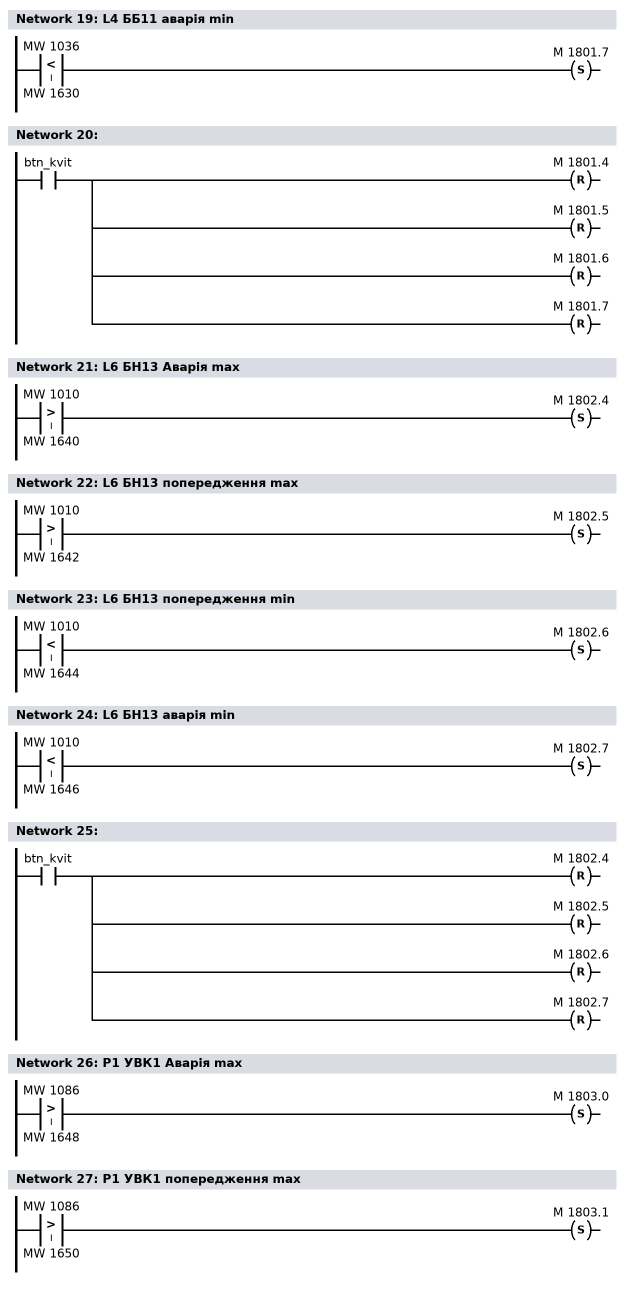
NETWORK
TITLE = L4 ББ11 аварія min
      L     MW 1036;
      L     MW 1630;
      <I;
      S     M 1801.7;
NETWORK
TITLE =
      A     "btn_kvit";
      R     M 1801.4;
      R     M 1801.5;
      R     M 1801.6;
      R     M 1801.7;
NETWORK
TITLE = L6 БН13 Аварія max
//*************************************************
      L     MW 1010;
      L     MW 1640;
      >I;
      S     M 1802.4;
NETWORK
TITLE = L6 БН13 попередження max
      L     MW 1010;
      L     MW 1642;
      >I;
      S     M 1802.5;
NETWORK
TITLE = L6 БН13 попередження min
      L     MW 1010;
      L     MW 1644;
      <I;
      S     M 1802.6;
NETWORK
TITLE = L6 БН13 аварія min
      L     MW 1010;
      L     MW 1646;
      <I;
      S     M 1802.7;
NETWORK
TITLE =
      A     "btn_kvit";
      R     M 1802.4;
      R     M 1802.5;
      R     M 1802.6;
      R     M 1802.7;
NETWORK
TITLE = P1 УВК1 Аварія max
//*************************************************
      L     MW 1086;
      L     MW 1648;
      >I;
      S     M 1803.0;
NETWORK
TITLE = P1 УВК1 попередження max
      L     MW 1086;
      L     MW 1650;
      >I;
      S     M 1803.1;
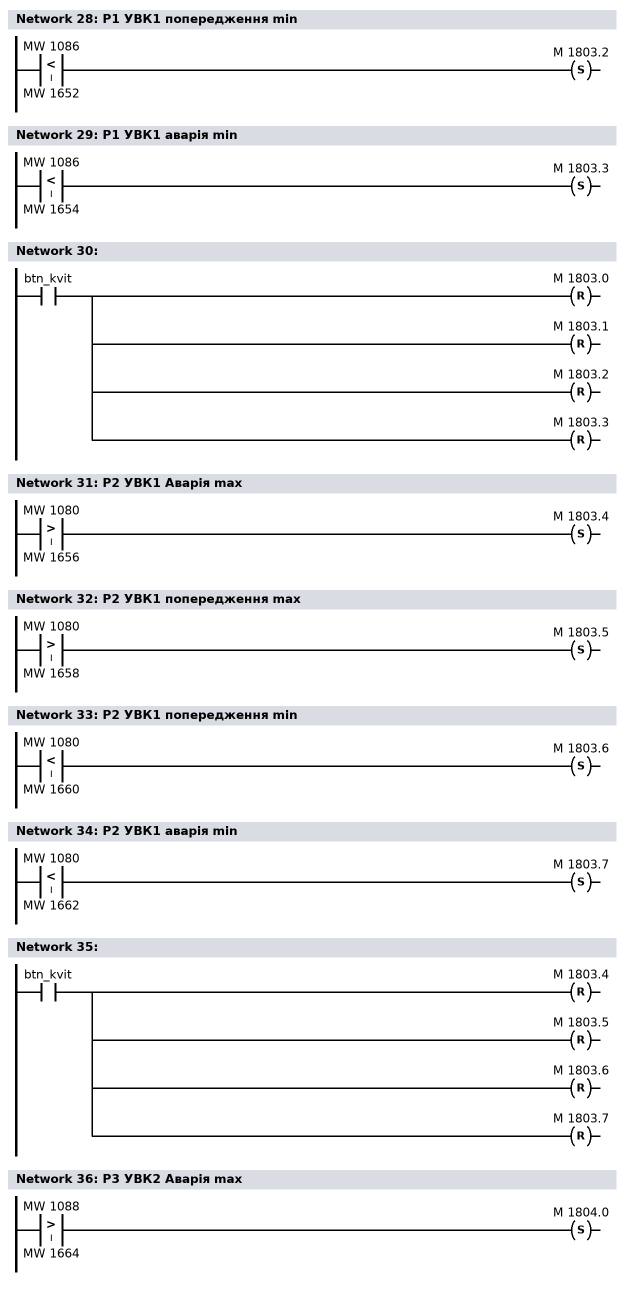
NETWORK
TITLE = P1 УВК1 попередження min
      L     MW 1086;
      L     MW 1652;
      <I;
      S     M 1803.2;
NETWORK
TITLE = P1 УВК1 аварія min
      L     MW 1086;
      L     MW 1654;
      <I;
      S     M 1803.3;
NETWORK
TITLE =
      A     "btn_kvit";
      R     M 1803.0;
      R     M 1803.1;
      R     M 1803.2;
      R     M 1803.3;
NETWORK
TITLE = P2 УВК1 Аварія max
//*************************************************
      L     MW 1080;
      L     MW 1656;
      >I;
      S     M 1803.4;
NETWORK
TITLE = P2 УВК1 попередження max
      L     MW 1080;
      L     MW 1658;
      >I;
      S     M 1803.5;
NETWORK
TITLE = P2 УВК1 попередження min
      L     MW 1080;
      L     MW 1660;
      <I;
      S     M 1803.6;
NETWORK
TITLE = P2 УВК1 аварія min
      L     MW 1080;
      L     MW 1662;
      <I;
      S     M 1803.7;
NETWORK
TITLE =
      A     "btn_kvit";
      R     M 1803.4;
      R     M 1803.5;
      R     M 1803.6;
      R     M 1803.7;
NETWORK
TITLE = P3 УВК2 Аварія max
//*************************************************
      L     MW 1088;
      L     MW 1664;
      >I;
      S     M 1804.0;
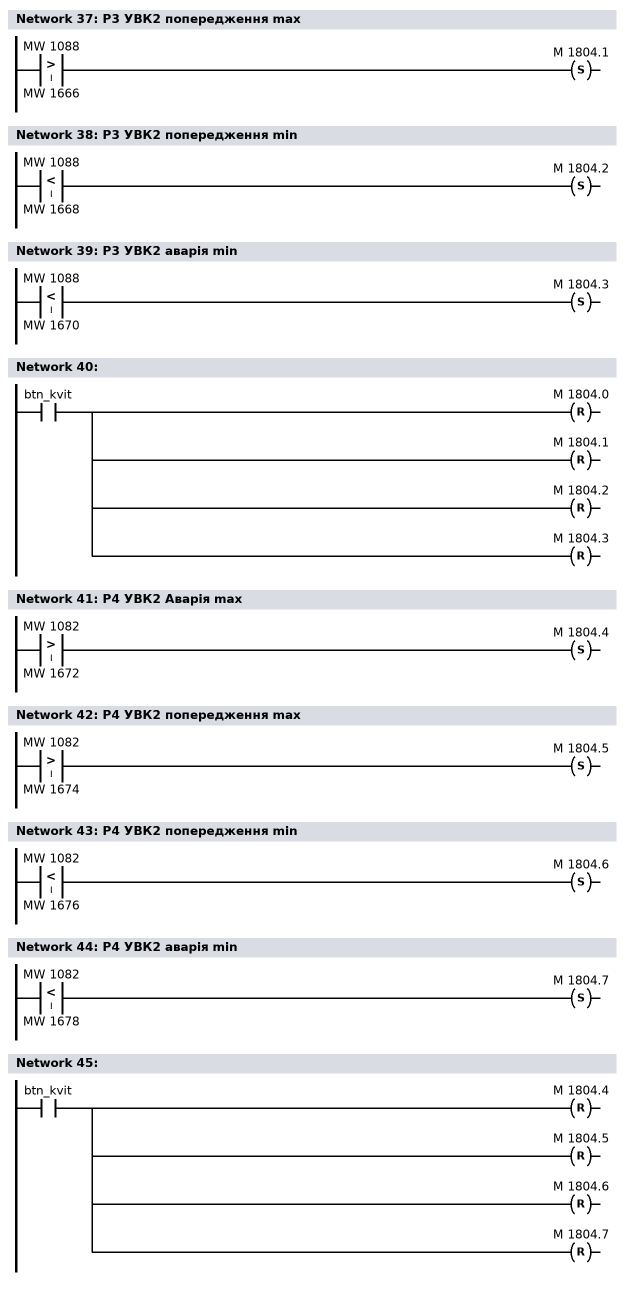
NETWORK
TITLE = P3 УВК2 попередження max
      L     MW 1088;
      L     MW 1666;
      >I;
      S     M 1804.1;
NETWORK
TITLE = P3 УВК2 попередження min
      L     MW 1088;
      L     MW 1668;
      <I;
      S     M 1804.2;
NETWORK
TITLE = P3 УВК2 аварія min
      L     MW 1088;
      L     MW 1670;
      <I;
      S     M 1804.3;
NETWORK
TITLE =
      A     "btn_kvit";
      R     M 1804.0;
      R     M 1804.1;
      R     M 1804.2;
      R     M 1804.3;
NETWORK
TITLE = P4 УВК2 Аварія max
//*************************************************
      L     MW 1082;
      L     MW 1672;
      >I;
      S     M 1804.4;
NETWORK
TITLE = P4 УВК2 попередження max
      L     MW 1082;
      L     MW 1674;
      >I;
      S     M 1804.5;
NETWORK
TITLE = P4 УВК2 попередження min
      L     MW 1082;
      L     MW 1676;
      <I;
      S     M 1804.6;
NETWORK
TITLE = P4 УВК2 аварія min
      L     MW 1082;
      L     MW 1678;
      <I;
      S     M 1804.7;
NETWORK
TITLE =
      A     "btn_kvit";
      R     M 1804.4;
      R     M 1804.5;
      R     M 1804.6;
      R     M 1804.7;
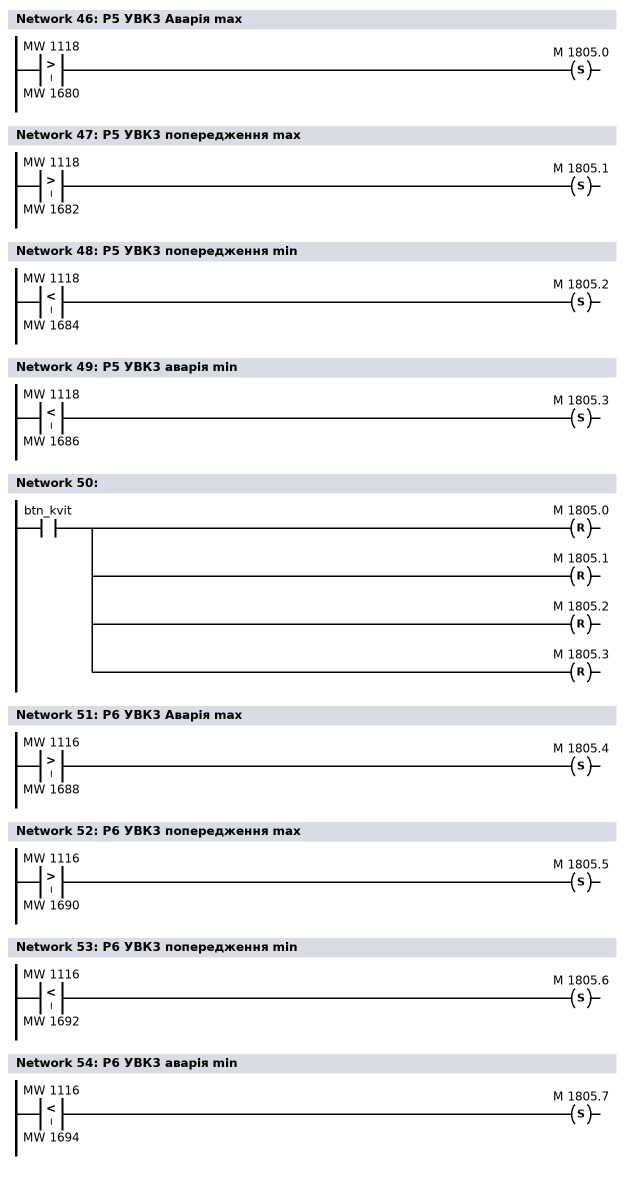
NETWORK
TITLE = P5 УВК3 Аварія max
//*************************************************
      L     MW 1118;
      L     MW 1680;
      >I;
      S     M 1805.0;
NETWORK
TITLE = P5 УВК3 попередження max
      L     MW 1118;
      L     MW 1682;
      >I;
      S     M 1805.1;
NETWORK
TITLE = P5 УВК3 попередження min
      L     MW 1118;
      L     MW 1684;
      <I;
      S     M 1805.2;
NETWORK
TITLE = P5 УВК3 аварія min
      L     MW 1118;
      L     MW 1686;
      <I;
      S     M 1805.3;
NETWORK
TITLE =
      A     "btn_kvit";
      R     M 1805.0;
      R     M 1805.1;
      R     M 1805.2;
      R     M 1805.3;
NETWORK
TITLE = P6 УВК3 Аварія max
//*************************************************
      L     MW 1116;
      L     MW 1688;
      >I;
      S     M 1805.4;
NETWORK
TITLE = P6 УВК3 попередження max
      L     MW 1116;
      L     MW 1690;
      >I;
      S     M 1805.5;
NETWORK
TITLE = P6 УВК3 попередження min
      L     MW 1116;
      L     MW 1692;
      <I;
      S     M 1805.6;
NETWORK
TITLE = P6 УВК3 аварія min
      L     MW 1116;
      L     MW 1694;
      <I;
      S     M 1805.7;
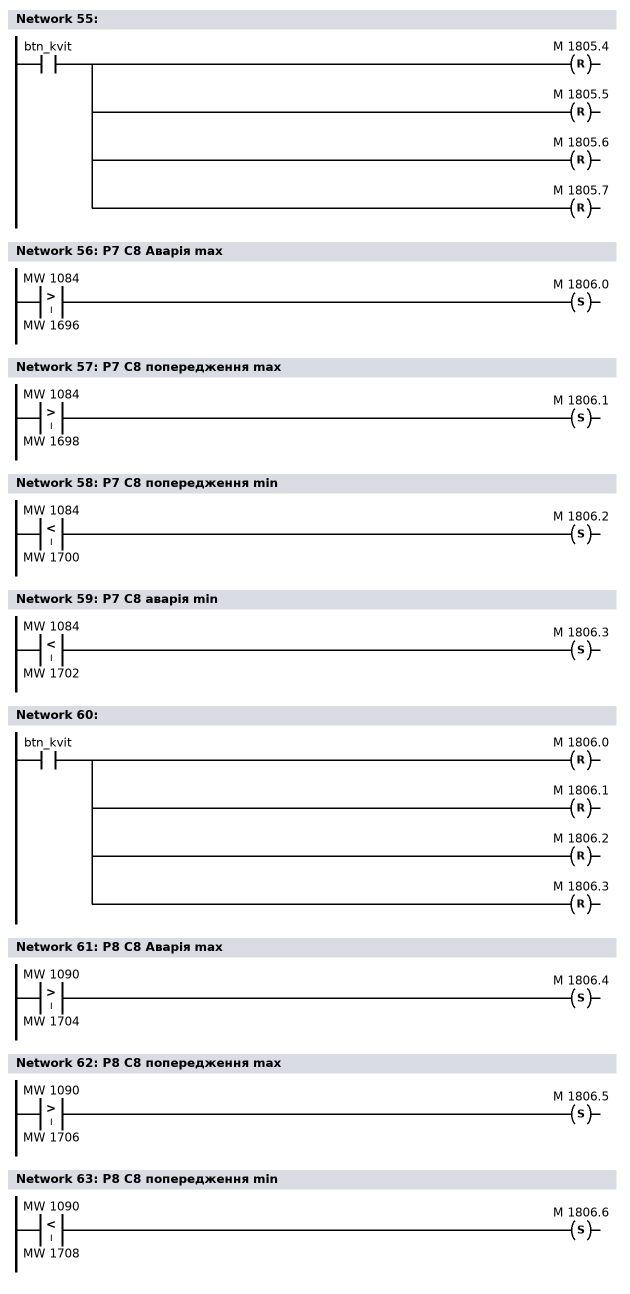
NETWORK
TITLE =
      A     "btn_kvit";
      R     M 1805.4;
      R     M 1805.5;
      R     M 1805.6;
      R     M 1805.7;
NETWORK
TITLE = P7 С8 Аварія max
//*************************************************
      L     MW 1084;
      L     MW 1696;
      >I;
      S     M 1806.0;
NETWORK
TITLE = P7 С8 попередження max
      L     MW 1084;
      L     MW 1698;
      >I;
      S     M 1806.1;
NETWORK
TITLE = P7 С8 попередження min
      L     MW 1084;
      L     MW 1700;
      <I;
      S     M 1806.2;
NETWORK
TITLE = P7 С8 аварія min
      L     MW 1084;
      L     MW 1702;
      <I;
      S     M 1806.3;
NETWORK
TITLE =
      A     "btn_kvit";
      R     M 1806.0;
      R     M 1806.1;
      R     M 1806.2;
      R     M 1806.3;
NETWORK
TITLE = P8 С8 Аварія max
//*************************************************
      L     MW 1090;
      L     MW 1704;
      >I;
      S     M 1806.4;
NETWORK
TITLE = P8 С8 попередження max
      L     MW 1090;
      L     MW 1706;
      >I;
      S     M 1806.5;
NETWORK
TITLE = P8 С8 попередження min
      L     MW 1090;
      L     MW 1708;
      <I;
      S     M 1806.6;
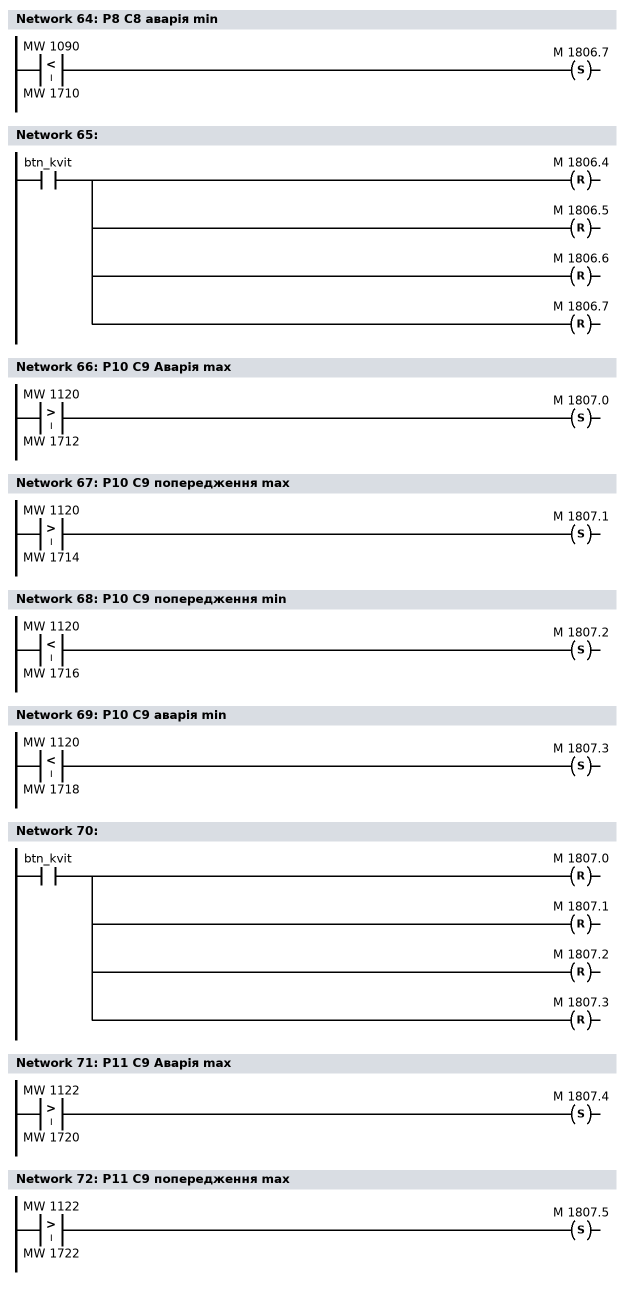
NETWORK
TITLE = P8 С8 аварія min
      L     MW 1090;
      L     MW 1710;
      <I;
      S     M 1806.7;
NETWORK
TITLE =
      A     "btn_kvit";
      R     M 1806.4;
      R     M 1806.5;
      R     M 1806.6;
      R     M 1806.7;
NETWORK
TITLE = P10 С9 Аварія max
//*************************************************
      L     MW 1120;
      L     MW 1712;
      >I;
      S     M 1807.0;
NETWORK
TITLE = P10 С9 попередження max
      L     MW 1120;
      L     MW 1714;
      >I;
      S     M 1807.1;
NETWORK
TITLE = P10 С9 попередження min
      L     MW 1120;
      L     MW 1716;
      <I;
      S     M 1807.2;
NETWORK
TITLE = P10 С9 аварія min
      L     MW 1120;
      L     MW 1718;
      <I;
      S     M 1807.3;
NETWORK
TITLE =
      A     "btn_kvit";
      R     M 1807.0;
      R     M 1807.1;
      R     M 1807.2;
      R     M 1807.3;
NETWORK
TITLE = P11 С9 Аварія max
//*************************************************
      L     MW 1122;
      L     MW 1720;
      >I;
      S     M 1807.4;
NETWORK
TITLE = P11 С9 попередження max
      L     MW 1122;
      L     MW 1722;
      >I;
      S     M 1807.5;
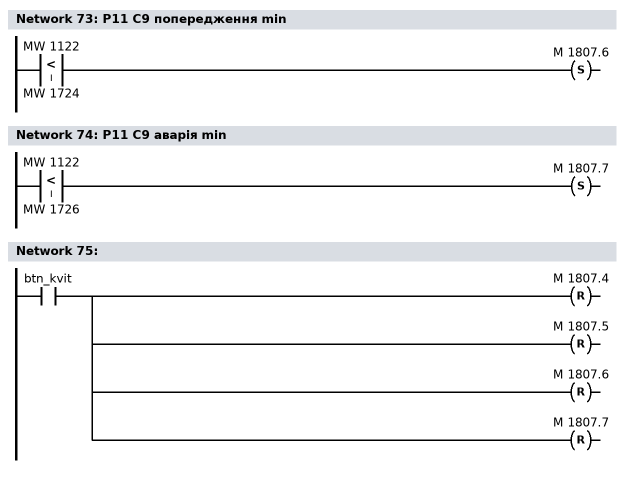
NETWORK
TITLE = P11 С9 попередження min
      L     MW 1122;
      L     MW 1724;
      <I;
      S     M 1807.6;
NETWORK
TITLE = P11 С9 аварія min
      L     MW 1122;
      L     MW 1726;
      <I;
      S     M 1807.7;
NETWORK
TITLE =
      A     "btn_kvit";
      R     M 1807.4;
      R     M 1807.5;
      R     M 1807.6;
      R     M 1807.7;
END_FUNCTION_BLOCK

// FB 58: know-how protected block, not included

FUNCTION "DO_MANUAL" : VOID	// FC 1
VERSION : 0.1
VAR_INPUT
  MANUAL : BOOL ;
  PUSK : BOOL ;
  STOP : BOOL ;
END_VAR
VAR_OUTPUT
  M_DO : BOOL ;
END_VAR
BEGIN
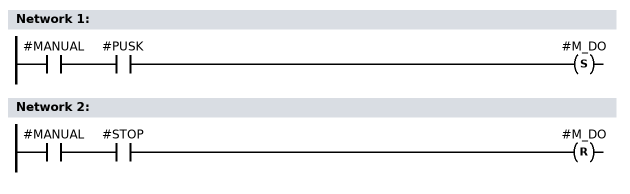
NETWORK
TITLE =
      A     #MANUAL;
      A     #PUSK;
      S     #M_DO;
NETWORK
TITLE =
      A     #MANUAL;
      A     #STOP;
      R     #M_DO;
END_FUNCTION

// FC 105: know-how protected block, not included

// FC 106: know-how protected block, not included

DATA_BLOCK DB 2
VERSION : 0.1
"MD_to_MW"
BEGIN
END_DATA_BLOCK

DATA_BLOCK DB 3
VERSION : 0.0
"DO_Control"
BEGIN
END_DATA_BLOCK

DATA_BLOCK DB 4
VERSION : 0.1
"DI_DO_STATE"
BEGIN
END_DATA_BLOCK

DATA_BLOCK DB 6
VERSION : 0.0
"dat_alm"
BEGIN
END_DATA_BLOCK

DATA_BLOCK DB 14
AUTHOR : SIMATIC
FAMILY : COM_FUNC
VERSION : 0.0
"GET"
BEGIN
END_DATA_BLOCK

DATA_BLOCK "COM"	// DB 100
VERSION : 0.1
  STRUCT
   dZN1_cur : REAL ;
   dUVK_nas1_cur : REAL ;
   dUVK_nas2_cur : REAL ;
   dUZ1_in : REAL ;
   dUZ1_out : REAL ;
   dPidsit_riv : REAL ;
   dVak_suknom1 : REAL ;
   dVak_suknom2 : REAL ;
   dVak_suknom3 : REAL ;
   dVak_suknom4 : REAL ;
   dVak_suknom5 : REAL ;
   dVak_suknom6 : REAL ;
   dVak_val1 : REAL ;
   dVak_val2 : REAL ;
   dVak_mok1 : REAL ;
   dVak_mok2 : REAL ;
   dVak_mok3 : REAL ;
   dVak_mok4 : REAL ;
   dVak_suh1 : REAL ;
   dVak_suh2 : REAL ;
   dVak_suh3 : REAL ;
   dVak_suh4 : REAL ;
   dVak_suh5 : REAL ;
   dVak_suh6 : REAL ;
   dVak_VN1 : REAL ;
   dVak_VN2 : REAL ;
   dVak_VN3 : REAL ;
   dVak_VN4 : REAL ;
   dVak_VN5 : REAL ;
   dBM8_riv : REAL ;
   dBO9_riv : REAL ;
   dBZ10_riv : REAL ;
   dBB11_riv : REAL ;
   dGauch_riv : REAL ;
   dNC32_riv : REAL ;
   dNC35_riv : REAL ;
   dPriamok_riv : REAL ;
   dGRG_riv : REAL ;
   task_ZNM12_re : REAL ;
   task_ZNM15_re : REAL ;
   dUVK1_in : REAL ;
   dUVK2_in : REAL ;
   dC8_in : REAL ;
   dUVK1_out : REAL ;
   dUVK2_out : REAL ;
   dC8_out : REAL ;
   dSUM_Pr_nya : REAL ;
   dConc1_nya : REAL ;
   dRiv_Skop : REAL ;
   dRiv_Bak_pid_nya : REAL ;
   dPr_uzloulov_in : REAL ;
   dMlyn_in : REAL ;
   dRiv_Bak_nap : REAL ;
   dMlyn_out : REAL ;
   dPr_uzloulov_out : REAL ;
   dRIV_NYA : REAL ;
  END_STRUCT ;	
BEGIN
END_DATA_BLOCK

DATA_BLOCK DB 101
VERSION : 0.0
"Dat_Filt"
BEGIN
END_DATA_BLOCK

DATA_BLOCK DB 102
VERSION : 0.0
"Dat_Filt"
BEGIN
END_DATA_BLOCK

DATA_BLOCK DB 103
VERSION : 0.0
"Dat_Filt"
BEGIN
END_DATA_BLOCK

DATA_BLOCK DB 104
VERSION : 0.0
"Dat_Filt"
BEGIN
END_DATA_BLOCK

DATA_BLOCK DB 105
VERSION : 0.0
"Dat_Filt"
BEGIN
END_DATA_BLOCK

DATA_BLOCK DB 106
VERSION : 0.0
"Dat_Filt"
BEGIN
END_DATA_BLOCK

DATA_BLOCK DB 107
VERSION : 0.0
"Dat_Filt"
BEGIN
END_DATA_BLOCK

DATA_BLOCK DB 108
VERSION : 0.0
"Dat_Filt"
BEGIN
END_DATA_BLOCK

DATA_BLOCK DB 109
VERSION : 0.0
"Dat_Filt"
BEGIN
END_DATA_BLOCK

DATA_BLOCK DB 110
VERSION : 0.0
"Dat_Filt"
BEGIN
END_DATA_BLOCK

DATA_BLOCK DB 111
VERSION : 0.0
"Dat_Filt"
BEGIN
END_DATA_BLOCK

DATA_BLOCK DB 112
VERSION : 0.0
"Dat_Filt"
BEGIN
END_DATA_BLOCK

DATA_BLOCK DB 113
VERSION : 0.0
"Dat_Filt"
BEGIN
END_DATA_BLOCK

DATA_BLOCK DB 114
VERSION : 0.0
"Dat_Filt"
BEGIN
END_DATA_BLOCK

DATA_BLOCK DB 115
VERSION : 0.0
"Dat_Filt"
BEGIN
END_DATA_BLOCK

DATA_BLOCK DB 116
VERSION : 0.0
"Dat_Filt"
BEGIN
END_DATA_BLOCK

DATA_BLOCK DB 117
VERSION : 0.0
"Dat_Filt"
BEGIN
END_DATA_BLOCK

DATA_BLOCK DB 118
VERSION : 0.0
"Dat_Filt"
BEGIN
END_DATA_BLOCK

DATA_BLOCK DB 119
VERSION : 0.0
"Dat_Filt"
BEGIN
END_DATA_BLOCK

DATA_BLOCK DB 120
VERSION : 0.0
"Dat_Filt"
BEGIN
END_DATA_BLOCK

DATA_BLOCK DB 121
VERSION : 0.0
"Dat_Filt"
BEGIN
END_DATA_BLOCK

DATA_BLOCK DB 122
VERSION : 0.0
"Dat_Filt"
BEGIN
END_DATA_BLOCK

DATA_BLOCK DB 123
VERSION : 0.0
"Dat_Filt"
BEGIN
END_DATA_BLOCK

DATA_BLOCK DB 124
VERSION : 0.0
"Dat_Filt"
BEGIN
END_DATA_BLOCK

DATA_BLOCK DB 125
VERSION : 0.0
"Dat_Filt"
BEGIN
END_DATA_BLOCK

DATA_BLOCK DB 126
VERSION : 0.0
"Dat_Filt"
BEGIN
END_DATA_BLOCK

DATA_BLOCK DB 127
VERSION : 0.0
"Dat_Filt"
BEGIN
END_DATA_BLOCK

DATA_BLOCK DB 128
VERSION : 0.0
"Dat_Filt"
BEGIN
END_DATA_BLOCK

DATA_BLOCK DB 141
VERSION : 0.0
"Dat_Filt"
BEGIN
END_DATA_BLOCK

DATA_BLOCK DB 142
VERSION : 0.0
"Dat_Filt"
BEGIN
END_DATA_BLOCK

DATA_BLOCK DB 143
VERSION : 0.0
"Dat_Filt"
BEGIN
END_DATA_BLOCK

DATA_BLOCK DB 144
VERSION : 0.0
"Dat_Filt"
BEGIN
END_DATA_BLOCK

DATA_BLOCK DB 145
VERSION : 0.0
"Dat_Filt"
BEGIN
END_DATA_BLOCK

DATA_BLOCK DB 146
VERSION : 0.0
"Dat_Filt"
BEGIN
END_DATA_BLOCK

DATA_BLOCK DB 147
VERSION : 0.0
"Dat_Filt"
BEGIN
END_DATA_BLOCK

DATA_BLOCK DB 148
VERSION : 0.0
"Dat_Filt"
BEGIN
END_DATA_BLOCK

DATA_BLOCK DB 149
VERSION : 0.0
"Dat_Filt"
BEGIN
END_DATA_BLOCK

DATA_BLOCK DB 150
VERSION : 0.0
"Dat_Filt"
BEGIN
END_DATA_BLOCK

DATA_BLOCK DB 151
VERSION : 0.0
"Dat_Filt"
BEGIN
END_DATA_BLOCK

DATA_BLOCK DB 152
VERSION : 0.0
"Dat_Filt"
BEGIN
END_DATA_BLOCK

DATA_BLOCK DB 153
VERSION : 0.0
"Dat_Filt"
BEGIN
END_DATA_BLOCK

DATA_BLOCK DB 154
VERSION : 0.0
"Dat_Filt"
BEGIN
END_DATA_BLOCK

DATA_BLOCK DB 155
VERSION : 0.0
"Dat_Filt"
BEGIN
END_DATA_BLOCK

DATA_BLOCK DB 300
VERSION : 0.0
"PID_AO_control"
BEGIN
END_DATA_BLOCK

DATA_BLOCK DB 301
VERSION : 0.0
"PID_AO_control"
BEGIN
END_DATA_BLOCK

DATA_BLOCK DB 302
VERSION : 0.0
"PID_AO_control"
BEGIN
END_DATA_BLOCK

DATA_BLOCK "znm15_pid"	// DB 500
AUTHOR : SIMATIC
FAMILY : CONTROL
VERSION : 0.0
"TCONT_CP"
BEGIN
END_DATA_BLOCK

DATA_BLOCK "CV_dConc1_pid"	// DB 501
AUTHOR : SIMATIC
FAMILY : CONTROL
VERSION : 0.0
"TCONT_CP"
BEGIN
END_DATA_BLOCK

DATA_BLOCK "zadv_riv_nya"	// DB 502
AUTHOR : SIMATIC
FAMILY : CONTROL
VERSION : 0.0
"TCONT_CP"
BEGIN
END_DATA_BLOCK

ORGANIZATION_BLOCK "CYCL_EXC"	// OB 1
TITLE = "Main Program Sweep (Cycle)"
VERSION : 0.1
VAR_TEMP
  OB1_EV_CLASS : BYTE ;	//Bits 0-3 = 1 (Coming event), Bits 4-7 = 1 (Event class 1)
  OB1_SCAN_1 : BYTE ;	//1 (Cold restart scan 1 of OB 1), 3 (Scan 2-n of OB 1)
  OB1_PRIORITY : BYTE ;	//Priority of OB Execution
  OB1_OB_NUMBR : BYTE ;	//1 (Organization block 1, OB1)
  OB1_RESERVED_1 : BYTE ;	//Reserved for system
  OB1_RESERVED_2 : BYTE ;	//Reserved for system
  OB1_PREV_CYCLE : INT ;	//Cycle time of previous OB1 scan (milliseconds)
  OB1_MIN_CYCLE : INT ;	//Minimum cycle time of OB1 (milliseconds)
  OB1_MAX_CYCLE : INT ;	//Maximum cycle time of OB1 (milliseconds)
  OB1_DATE_TIME : DATE_AND_TIME ;	//Date and time OB1 started
  err_ZN1_cur : BOOL ;
  err_UVK1_cur : BOOL ;
  err_UVK2_cur : BOOL ;
  err_UZ1_in : BOOL ;
  err_UZ1_out : BOOL ;
  err_pidsit_riv : BOOL ;
  err_vak_suknom1 : BOOL ;
  err_vak_suknom2 : BOOL ;
  err_vak_suknom3 : BOOL ;
  err_vak_suknom4 : BOOL ;
  err_vak_suknom5 : BOOL ;
  err_vak_suknom6 : BOOL ;
  err_vak_val1 : BOOL ;
  err_vak_val2 : BOOL ;
  err_vak_mok1 : BOOL ;
  err_vak_mok2 : BOOL ;
  err_vak_mok3 : BOOL ;
  err_vak_mok4 : BOOL ;
  err_suh1 : BOOL ;
  err_suh2 : BOOL ;
  err_suh3 : BOOL ;
  err_suh4 : BOOL ;
  err_suh5 : BOOL ;
  err_suh6 : BOOL ;
  err_vak_VN1 : BOOL ;
  err_vak_VN2 : BOOL ;
  err_vak_VN3 : BOOL ;
  err_vak_VN4 : BOOL ;
  err_vak_VN5 : BOOL ;
  err_BM8_riv : BOOL ;
  err_BO9_riv : BOOL ;
  err_BZ10_riv : BOOL ;
  err_BB11_riv : BOOL ;
  err_Gauch_riv : BOOL ;
  err_NC32_riv : BOOL ;
  err_NC35_riv : BOOL ;
  err_Priamok_riv : BOOL ;
  err_GRG_riv : BOOL ;
  ZNM12_ret : WORD ;
  ZNM15_ret : WORD ;
  bipolar : BOOL ;
  err_dUVK1in : BOOL ;
  err_dUVK2in : BOOL ;
  err_dC8in : BOOL ;
  err_dUVK1out : BOOL ;
  err_dUVK2out : BOOL ;
  err_dC8out : BOOL ;
  err_dSumPR : BOOL ;
  err_dConc1 : BOOL ;
  err_dBakSkop : BOOL ;
  err_dBakpidNya : BOOL ;
  err_dMlyn_in : BOOL ;
  err_uzloulov_in : BOOL ;
  err_dMlyn_out : BOOL ;
  err_uzloulov_out : BOOL ;
  bypass : BOOL ;
  err_dRIV_NYA : BOOL ;
END_VAR
BEGIN
NETWORK
TITLE = Из ПЛК ДВГ берем 10 байт в ПЛК КИП (кнопки "ручний режим")
      A     M 100.3;
      =     L 33.0;
      BLD   103;
      BLD   9;
      =     L 38.0;
      CDB;
      OPN   DI 14;
      TAR2  LD 34;
      A     L 33.0;
      =     DIX 0.0;
      L     2;
      T     DIW 2;
      L     W#16#1002;
      T     DIW 8;
      L     10;
      T     DIW 10;
      L     0;
      T     DIW 12;
      L     P#M 2000.0;
      T     DID 14;
      L     W#16#1002;
      T     DIW 48;
      L     10;
      T     DIW 50;
      L     0;
      T     DIW 52;
      L     P#M 6000.0;
      T     DID 54;
      LAR2  P#DBX 0.0;
      UC    "GET";
      LAR2  LD 34;
      CDB;
      BLD   10;
      NOP   0;
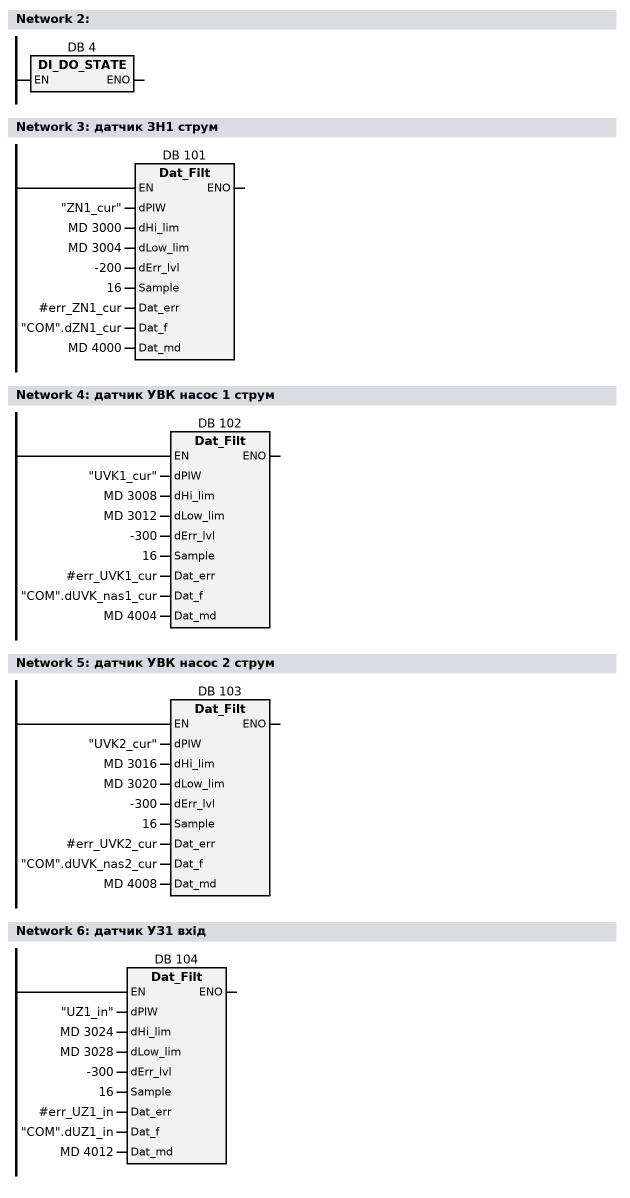
NETWORK
TITLE =
      CALL  "DI_DO_STATE" , DB 4;
      NOP   0;
NETWORK
TITLE = датчик ЗН1 струм  
      CALL  "Dat_Filt" , DB 101 (
           dPIW                     := "ZN1_cur",
           dHi_lim                  := MD 3000,
           dLow_lim                 := MD 3004,
           dErr_lvl                 := -200,
           Sample                   := 16,
           Dat_err                  := #err_ZN1_cur,
           Dat_f                    := "COM".dZN1_cur,
           Dat_md                   := MD 4000);
      NOP   0;
NETWORK
TITLE = датчик УВК насос 1 струм 
      CALL  "Dat_Filt" , DB 102 (
           dPIW                     := "UVK1_cur",
           dHi_lim                  := MD 3008,
           dLow_lim                 := MD 3012,
           dErr_lvl                 := -300,
           Sample                   := 16,
           Dat_err                  := #err_UVK1_cur,
           Dat_f                    := "COM".dUVK_nas1_cur,
           Dat_md                   := MD 4004);
      NOP   0;
NETWORK
TITLE = датчик УВК насос 2 струм 
      CALL  "Dat_Filt" , DB 103 (
           dPIW                     := "UVK2_cur",
           dHi_lim                  := MD 3016,
           dLow_lim                 := MD 3020,
           dErr_lvl                 := -300,
           Sample                   := 16,
           Dat_err                  := #err_UVK2_cur,
           Dat_f                    := "COM".dUVK_nas2_cur,
           Dat_md                   := MD 4008);
      NOP   0;
NETWORK
TITLE = датчик УЗ1 вхід
      CALL  "Dat_Filt" , DB 104 (
           dPIW                     := "UZ1_in",
           dHi_lim                  := MD 3024,
           dLow_lim                 := MD 3028,
           dErr_lvl                 := -300,
           Sample                   := 16,
           Dat_err                  := #err_UZ1_in,
           Dat_f                    := "COM".dUZ1_in,
           Dat_md                   := MD 4012);
      NOP   0;
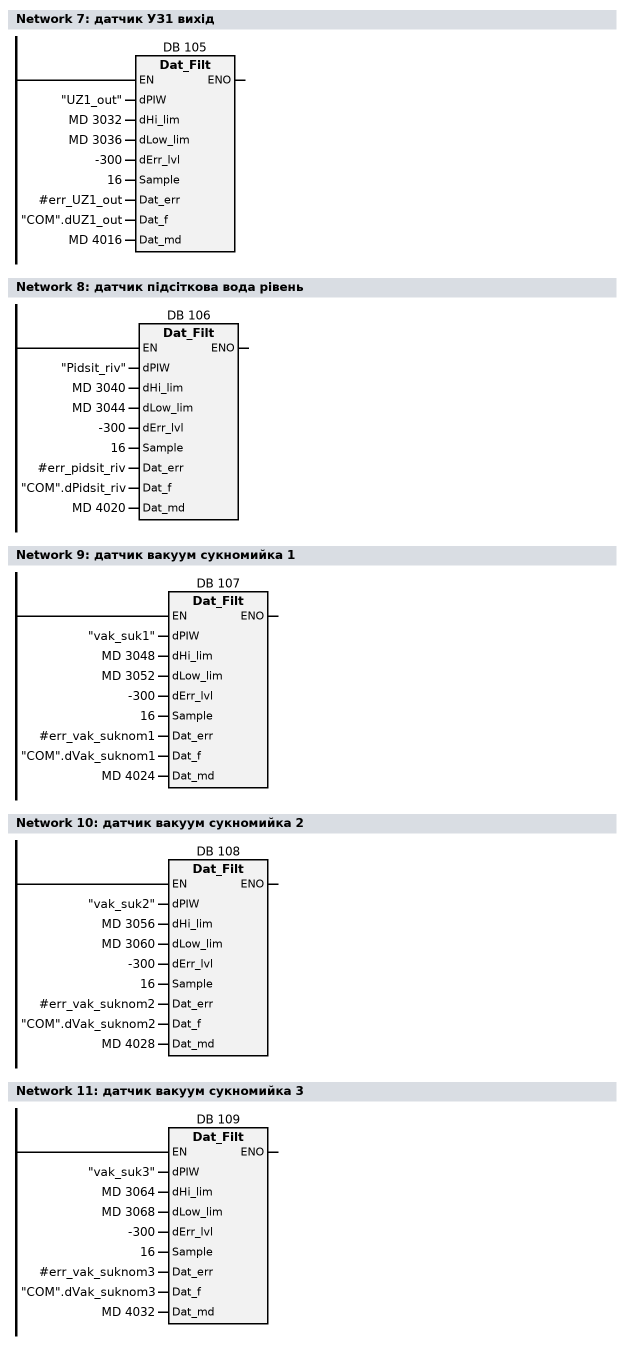
NETWORK
TITLE = датчик УЗ1 вихід
      CALL  "Dat_Filt" , DB 105 (
           dPIW                     := "UZ1_out",
           dHi_lim                  := MD 3032,
           dLow_lim                 := MD 3036,
           dErr_lvl                 := -300,
           Sample                   := 16,
           Dat_err                  := #err_UZ1_out,
           Dat_f                    := "COM".dUZ1_out,
           Dat_md                   := MD 4016);
      NOP   0;
NETWORK
TITLE = датчик підсіткова вода рівень
      CALL  "Dat_Filt" , DB 106 (
           dPIW                     := "Pidsit_riv",
           dHi_lim                  := MD 3040,
           dLow_lim                 := MD 3044,
           dErr_lvl                 := -300,
           Sample                   := 16,
           Dat_err                  := #err_pidsit_riv,
           Dat_f                    := "COM".dPidsit_riv,
           Dat_md                   := MD 4020);
      NOP   0;
NETWORK
TITLE = датчик вакуум сукномийка 1
      CALL  "Dat_Filt" , DB 107 (
           dPIW                     := "vak_suk1",
           dHi_lim                  := MD 3048,
           dLow_lim                 := MD 3052,
           dErr_lvl                 := -300,
           Sample                   := 16,
           Dat_err                  := #err_vak_suknom1,
           Dat_f                    := "COM".dVak_suknom1,
           Dat_md                   := MD 4024);
      NOP   0;
NETWORK
TITLE = датчик вакуум сукномийка 2
      CALL  "Dat_Filt" , DB 108 (
           dPIW                     := "vak_suk2",
           dHi_lim                  := MD 3056,
           dLow_lim                 := MD 3060,
           dErr_lvl                 := -300,
           Sample                   := 16,
           Dat_err                  := #err_vak_suknom2,
           Dat_f                    := "COM".dVak_suknom2,
           Dat_md                   := MD 4028);
      NOP   0;
NETWORK
TITLE = датчик вакуум сукномийка 3
      CALL  "Dat_Filt" , DB 109 (
           dPIW                     := "vak_suk3",
           dHi_lim                  := MD 3064,
           dLow_lim                 := MD 3068,
           dErr_lvl                 := -300,
           Sample                   := 16,
           Dat_err                  := #err_vak_suknom3,
           Dat_f                    := "COM".dVak_suknom3,
           Dat_md                   := MD 4032);
      NOP   0;
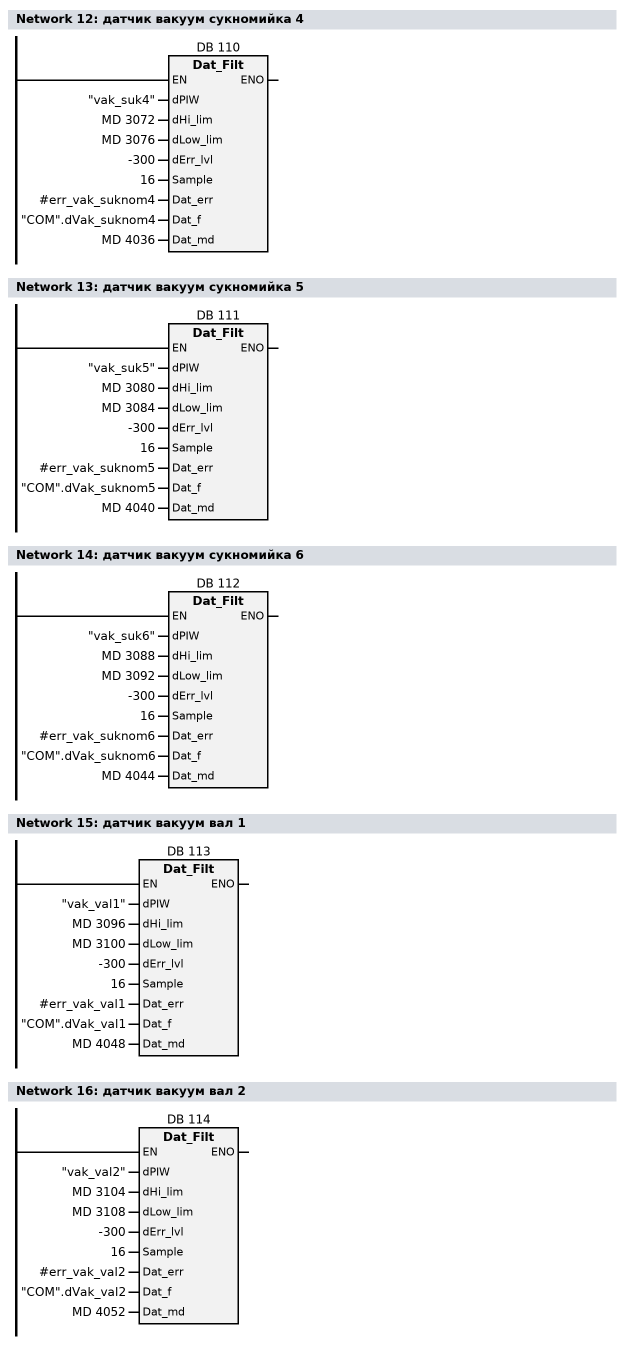
NETWORK
TITLE = датчик вакуум сукномийка 4
      CALL  "Dat_Filt" , DB 110 (
           dPIW                     := "vak_suk4",
           dHi_lim                  := MD 3072,
           dLow_lim                 := MD 3076,
           dErr_lvl                 := -300,
           Sample                   := 16,
           Dat_err                  := #err_vak_suknom4,
           Dat_f                    := "COM".dVak_suknom4,
           Dat_md                   := MD 4036);
      NOP   0;
NETWORK
TITLE = датчик вакуум сукномийка 5
      CALL  "Dat_Filt" , DB 111 (
           dPIW                     := "vak_suk5",
           dHi_lim                  := MD 3080,
           dLow_lim                 := MD 3084,
           dErr_lvl                 := -300,
           Sample                   := 16,
           Dat_err                  := #err_vak_suknom5,
           Dat_f                    := "COM".dVak_suknom5,
           Dat_md                   := MD 4040);
      NOP   0;
NETWORK
TITLE = датчик вакуум сукномийка 6
      CALL  "Dat_Filt" , DB 112 (
           dPIW                     := "vak_suk6",
           dHi_lim                  := MD 3088,
           dLow_lim                 := MD 3092,
           dErr_lvl                 := -300,
           Sample                   := 16,
           Dat_err                  := #err_vak_suknom6,
           Dat_f                    := "COM".dVak_suknom6,
           Dat_md                   := MD 4044);
      NOP   0;
NETWORK
TITLE = датчик вакуум вал 1
      CALL  "Dat_Filt" , DB 113 (
           dPIW                     := "vak_val1",
           dHi_lim                  := MD 3096,
           dLow_lim                 := MD 3100,
           dErr_lvl                 := -300,
           Sample                   := 16,
           Dat_err                  := #err_vak_val1,
           Dat_f                    := "COM".dVak_val1,
           Dat_md                   := MD 4048);
      NOP   0;
NETWORK
TITLE = датчик вакуум вал 2
      CALL  "Dat_Filt" , DB 114 (
           dPIW                     := "vak_val2",
           dHi_lim                  := MD 3104,
           dLow_lim                 := MD 3108,
           dErr_lvl                 := -300,
           Sample                   := 16,
           Dat_err                  := #err_vak_val2,
           Dat_f                    := "COM".dVak_val2,
           Dat_md                   := MD 4052);
      NOP   0;
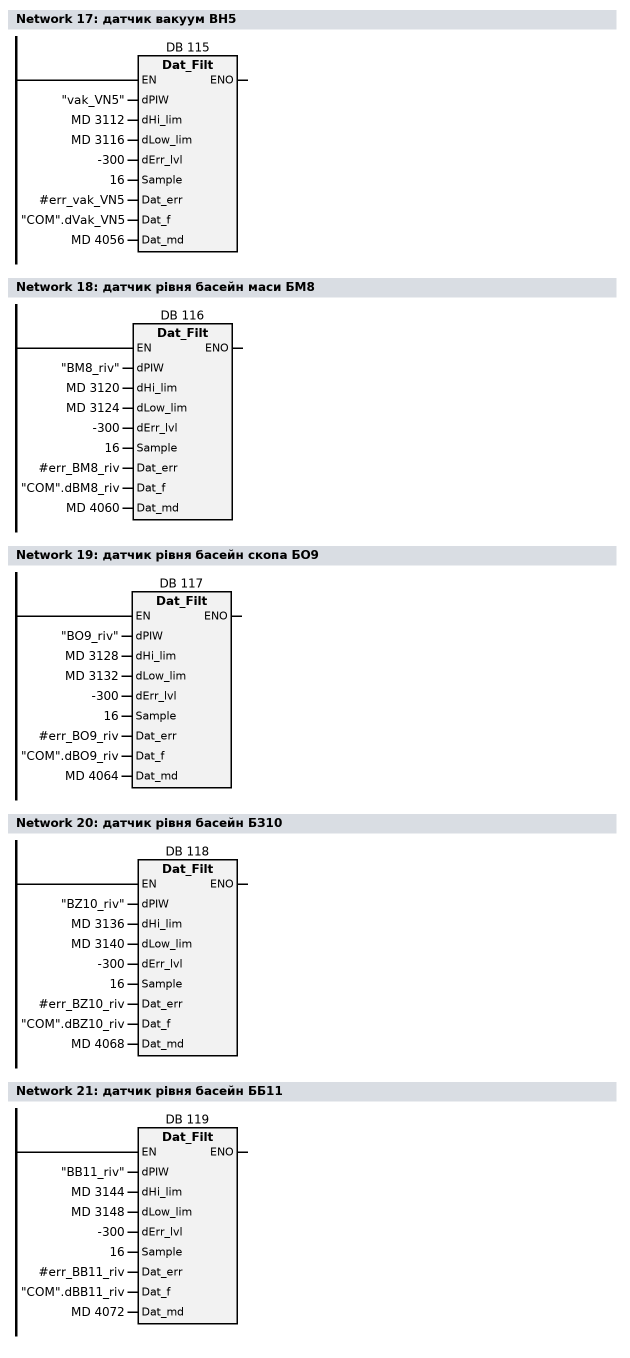
NETWORK
TITLE = датчик вакуум ВН5
      CALL  "Dat_Filt" , DB 115 (
           dPIW                     := "vak_VN5",
           dHi_lim                  := MD 3112,
           dLow_lim                 := MD 3116,
           dErr_lvl                 := -300,
           Sample                   := 16,
           Dat_err                  := #err_vak_VN5,
           Dat_f                    := "COM".dVak_VN5,
           Dat_md                   := MD 4056);
      NOP   0;
NETWORK
TITLE = датчик рівня басейн маси БМ8
      CALL  "Dat_Filt" , DB 116 (
           dPIW                     := "BM8_riv",
           dHi_lim                  := MD 3120,
           dLow_lim                 := MD 3124,
           dErr_lvl                 := -300,
           Sample                   := 16,
           Dat_err                  := #err_BM8_riv,
           Dat_f                    := "COM".dBM8_riv,
           Dat_md                   := MD 4060);
      NOP   0;
NETWORK
TITLE = датчик рівня басейн скопа БО9
      CALL  "Dat_Filt" , DB 117 (
           dPIW                     := "BO9_riv",
           dHi_lim                  := MD 3128,
           dLow_lim                 := MD 3132,
           dErr_lvl                 := -300,
           Sample                   := 16,
           Dat_err                  := #err_BO9_riv,
           Dat_f                    := "COM".dBO9_riv,
           Dat_md                   := MD 4064);
      NOP   0;
NETWORK
TITLE = датчик рівня басейн БЗ10
      CALL  "Dat_Filt" , DB 118 (
           dPIW                     := "BZ10_riv",
           dHi_lim                  := MD 3136,
           dLow_lim                 := MD 3140,
           dErr_lvl                 := -300,
           Sample                   := 16,
           Dat_err                  := #err_BZ10_riv,
           Dat_f                    := "COM".dBZ10_riv,
           Dat_md                   := MD 4068);
      NOP   0;
NETWORK
TITLE = датчик рівня басейн ББ11
      CALL  "Dat_Filt" , DB 119 (
           dPIW                     := "BB11_riv",
           dHi_lim                  := MD 3144,
           dLow_lim                 := MD 3148,
           dErr_lvl                 := -300,
           Sample                   := 16,
           Dat_err                  := #err_BB11_riv,
           Dat_f                    := "COM".dBB11_riv,
           Dat_md                   := MD 4072);
      NOP   0;
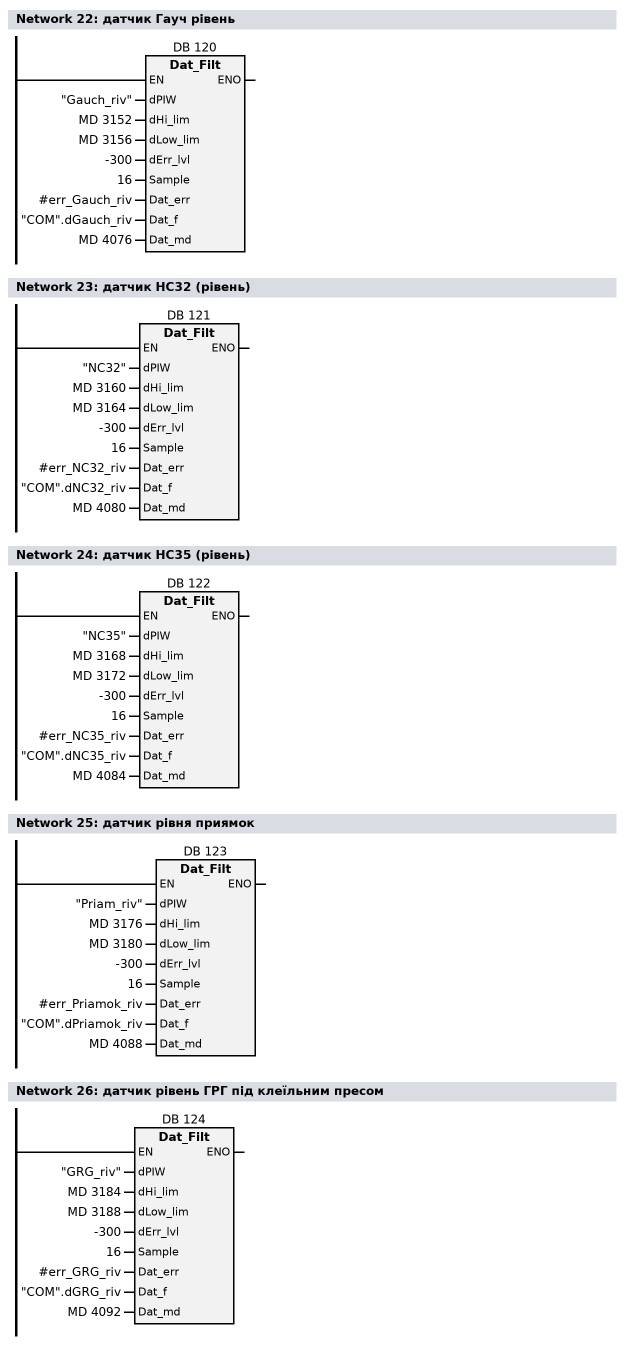
NETWORK
TITLE = датчик Гауч рівень
      CALL  "Dat_Filt" , DB 120 (
           dPIW                     := "Gauch_riv",
           dHi_lim                  := MD 3152,
           dLow_lim                 := MD 3156,
           dErr_lvl                 := -300,
           Sample                   := 16,
           Dat_err                  := #err_Gauch_riv,
           Dat_f                    := "COM".dGauch_riv,
           Dat_md                   := MD 4076);
      NOP   0;
NETWORK
TITLE = датчик НС32 (рівень)
      CALL  "Dat_Filt" , DB 121 (
           dPIW                     := "NC32",
           dHi_lim                  := MD 3160,
           dLow_lim                 := MD 3164,
           dErr_lvl                 := -300,
           Sample                   := 16,
           Dat_err                  := #err_NC32_riv,
           Dat_f                    := "COM".dNC32_riv,
           Dat_md                   := MD 4080);
      NOP   0;
NETWORK
TITLE = датчик НС35 (рівень)
      CALL  "Dat_Filt" , DB 122 (
           dPIW                     := "NC35",
           dHi_lim                  := MD 3168,
           dLow_lim                 := MD 3172,
           dErr_lvl                 := -300,
           Sample                   := 16,
           Dat_err                  := #err_NC35_riv,
           Dat_f                    := "COM".dNC35_riv,
           Dat_md                   := MD 4084);
      NOP   0;
NETWORK
TITLE = датчик рівня приямок
      CALL  "Dat_Filt" , DB 123 (
           dPIW                     := "Priam_riv",
           dHi_lim                  := MD 3176,
           dLow_lim                 := MD 3180,
           dErr_lvl                 := -300,
           Sample                   := 16,
           Dat_err                  := #err_Priamok_riv,
           Dat_f                    := "COM".dPriamok_riv,
           Dat_md                   := MD 4088);
      NOP   0;
NETWORK
TITLE = датчик рівень ГРГ під клеїльним пресом
      CALL  "Dat_Filt" , DB 124 (
           dPIW                     := "GRG_riv",
           dHi_lim                  := MD 3184,
           dLow_lim                 := MD 3188,
           dErr_lvl                 := -300,
           Sample                   := 16,
           Dat_err                  := #err_GRG_riv,
           Dat_f                    := "COM".dGRG_riv,
           Dat_md                   := MD 4092);
      NOP   0;
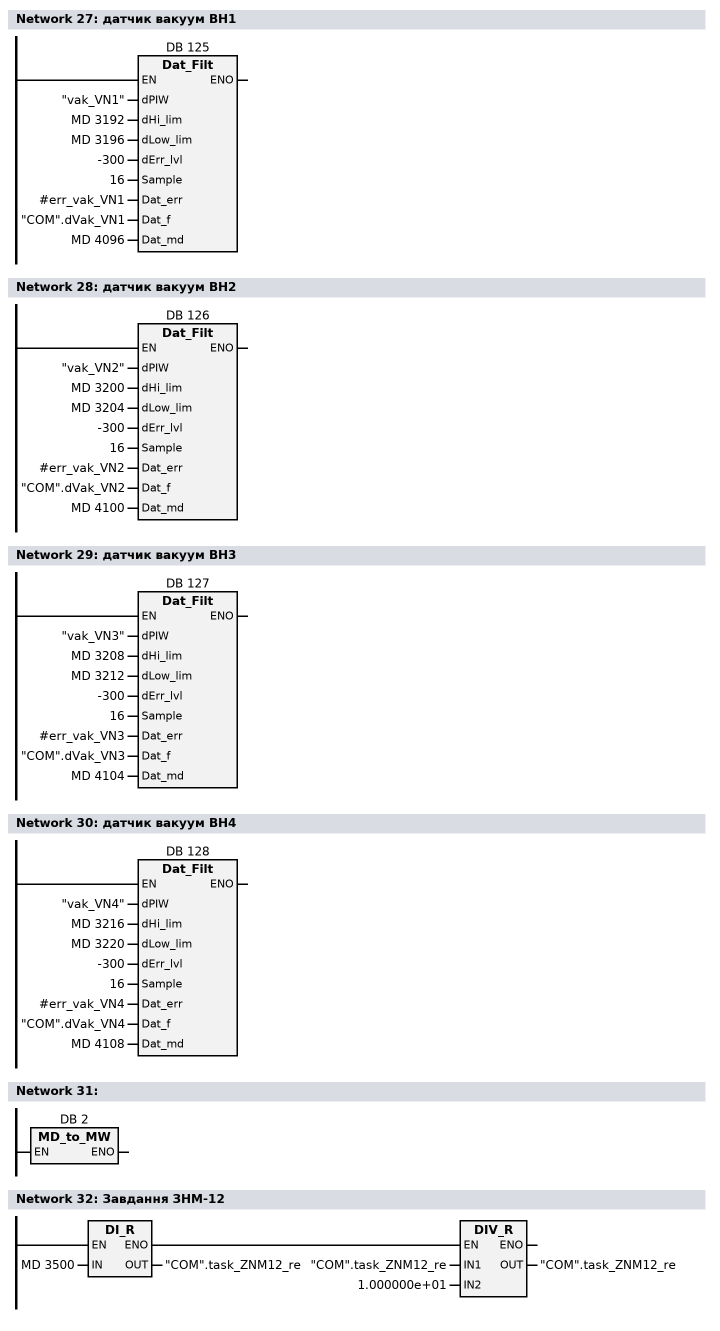
NETWORK
TITLE = датчик вакуум ВН1
      CALL  "Dat_Filt" , DB 125 (
           dPIW                     := "vak_VN1",
           dHi_lim                  := MD 3192,
           dLow_lim                 := MD 3196,
           dErr_lvl                 := -300,
           Sample                   := 16,
           Dat_err                  := #err_vak_VN1,
           Dat_f                    := "COM".dVak_VN1,
           Dat_md                   := MD 4096);
      NOP   0;
NETWORK
TITLE = датчик вакуум ВН2
      CALL  "Dat_Filt" , DB 126 (
           dPIW                     := "vak_VN2",
           dHi_lim                  := MD 3200,
           dLow_lim                 := MD 3204,
           dErr_lvl                 := -300,
           Sample                   := 16,
           Dat_err                  := #err_vak_VN2,
           Dat_f                    := "COM".dVak_VN2,
           Dat_md                   := MD 4100);
      NOP   0;
NETWORK
TITLE = датчик вакуум ВН3
      CALL  "Dat_Filt" , DB 127 (
           dPIW                     := "vak_VN3",
           dHi_lim                  := MD 3208,
           dLow_lim                 := MD 3212,
           dErr_lvl                 := -300,
           Sample                   := 16,
           Dat_err                  := #err_vak_VN3,
           Dat_f                    := "COM".dVak_VN3,
           Dat_md                   := MD 4104);
      NOP   0;
NETWORK
TITLE = датчик вакуум ВН4
      CALL  "Dat_Filt" , DB 128 (
           dPIW                     := "vak_VN4",
           dHi_lim                  := MD 3216,
           dLow_lim                 := MD 3220,
           dErr_lvl                 := -300,
           Sample                   := 16,
           Dat_err                  := #err_vak_VN4,
           Dat_f                    := "COM".dVak_VN4,
           Dat_md                   := MD 4108);
      NOP   0;
NETWORK
TITLE =
//Зборка блоку значень датчиків (і клапанів) для передачі по мережі
      CALL  "MD_to_MW" , DB 2;
      NOP   0;
NETWORK
TITLE = Завдання ЗНМ-12
//Завдання ЗНМ-12 в real
      A(;
      L     MD 3500;
      DTR;
      T     "COM".task_ZNM12_re;
      SET;
      SAVE;
      CLR;
      A     BR;
      );
      JNB   _001;
      L     "COM".task_ZNM12_re;
      L     1.000000e+01;
      /R;
      T     "COM".task_ZNM12_re;
_001: NOP   0;
NETWORK
TITLE = Завдання ЗНМ-12 записуємо в AO 1_1
      A(;
      A     #bipolar;
      =     L 33.0;
      BLD   103;
      CALL  "UNSCALE" (
           $1                       := "COM".task_ZNM12_re,
           $2                       := L#1120403456,
           $3                       := L#0,
           $4                       := L 33.0,
           $5                       := #ZNM12_ret,
           $6                       := P#M 4500.0);
      A     BR;
      );
      JNB   _002;
      L     MW 4500;
      T     "taskZNM12";
_002: NOP   0;
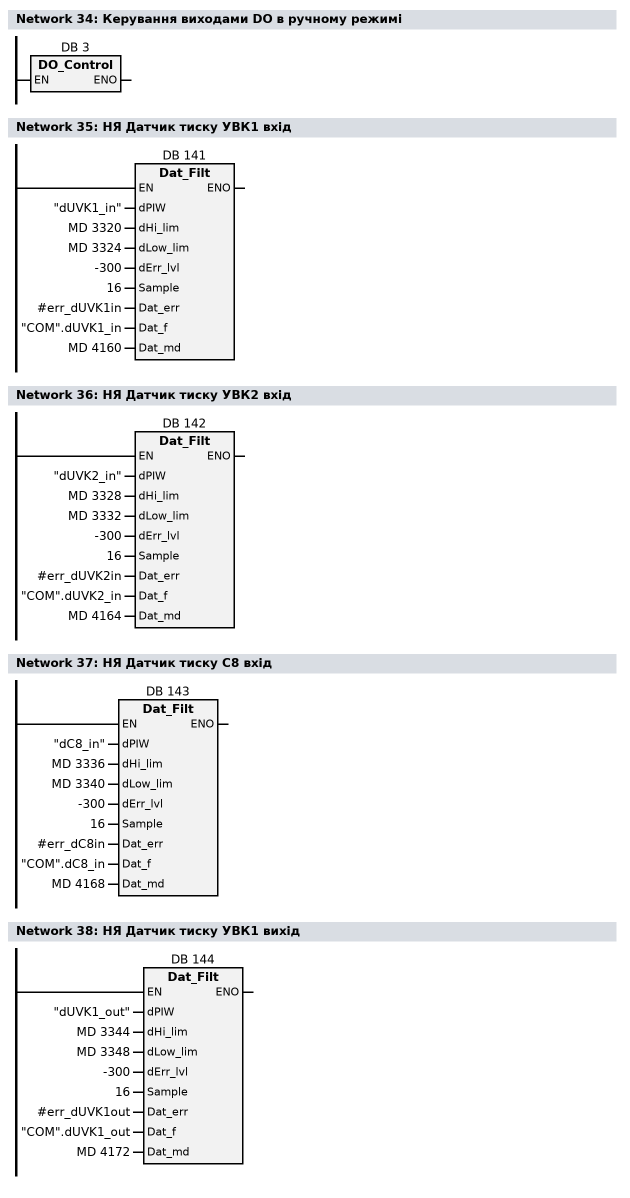
NETWORK
TITLE = Керування виходами DO в ручному режимі
      CALL  "DO_Control" , DB 3;
      NOP   0;
NETWORK
TITLE = НЯ Датчик тиску УВК1 вхід
//*******************************************************************************
      CALL  "Dat_Filt" , DB 141 (
           dPIW                     := "dUVK1_in",
           dHi_lim                  := MD 3320,
           dLow_lim                 := MD 3324,
           dErr_lvl                 := -300,
           Sample                   := 16,
           Dat_err                  := #err_dUVK1in,
           Dat_f                    := "COM".dUVK1_in,
           Dat_md                   := MD 4160);
      NOP   0;
NETWORK
TITLE = НЯ Датчик тиску УВК2 вхід
      CALL  "Dat_Filt" , DB 142 (
           dPIW                     := "dUVK2_in",
           dHi_lim                  := MD 3328,
           dLow_lim                 := MD 3332,
           dErr_lvl                 := -300,
           Sample                   := 16,
           Dat_err                  := #err_dUVK2in,
           Dat_f                    := "COM".dUVK2_in,
           Dat_md                   := MD 4164);
      NOP   0;
NETWORK
TITLE = НЯ Датчик тиску C8 вхід
      CALL  "Dat_Filt" , DB 143 (
           dPIW                     := "dC8_in",
           dHi_lim                  := MD 3336,
           dLow_lim                 := MD 3340,
           dErr_lvl                 := -300,
           Sample                   := 16,
           Dat_err                  := #err_dC8in,
           Dat_f                    := "COM".dC8_in,
           Dat_md                   := MD 4168);
      NOP   0;
NETWORK
TITLE = НЯ Датчик тиску УВК1 вихід
      CALL  "Dat_Filt" , DB 144 (
           dPIW                     := "dUVK1_out",
           dHi_lim                  := MD 3344,
           dLow_lim                 := MD 3348,
           dErr_lvl                 := -300,
           Sample                   := 16,
           Dat_err                  := #err_dUVK1out,
           Dat_f                    := "COM".dUVK1_out,
           Dat_md                   := MD 4172);
      NOP   0;
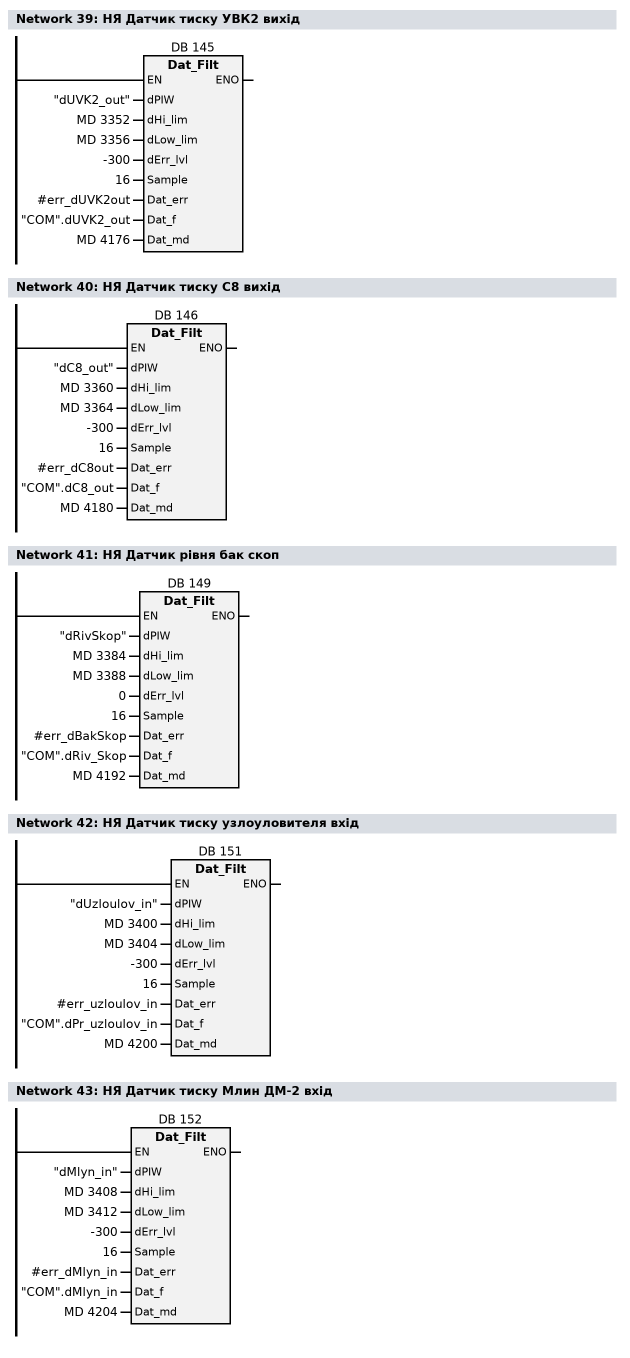
NETWORK
TITLE = НЯ Датчик тиску УВК2 вихід
      CALL  "Dat_Filt" , DB 145 (
           dPIW                     := "dUVK2_out",
           dHi_lim                  := MD 3352,
           dLow_lim                 := MD 3356,
           dErr_lvl                 := -300,
           Sample                   := 16,
           Dat_err                  := #err_dUVK2out,
           Dat_f                    := "COM".dUVK2_out,
           Dat_md                   := MD 4176);
      NOP   0;
NETWORK
TITLE = НЯ Датчик тиску C8 вихід
      CALL  "Dat_Filt" , DB 146 (
           dPIW                     := "dC8_out",
           dHi_lim                  := MD 3360,
           dLow_lim                 := MD 3364,
           dErr_lvl                 := -300,
           Sample                   := 16,
           Dat_err                  := #err_dC8out,
           Dat_f                    := "COM".dC8_out,
           Dat_md                   := MD 4180);
      NOP   0;
NETWORK
TITLE = НЯ Датчик рівня бак скоп
      CALL  "Dat_Filt" , DB 149 (
           dPIW                     := "dRivSkop",
           dHi_lim                  := MD 3384,
           dLow_lim                 := MD 3388,
           dErr_lvl                 := 0,
           Sample                   := 16,
           Dat_err                  := #err_dBakSkop,
           Dat_f                    := "COM".dRiv_Skop,
           Dat_md                   := MD 4192);
      NOP   0;
NETWORK
TITLE = НЯ Датчик тиску узлоуловителя вхід
      CALL  "Dat_Filt" , DB 151 (
           dPIW                     := "dUzloulov_in",
           dHi_lim                  := MD 3400,
           dLow_lim                 := MD 3404,
           dErr_lvl                 := -300,
           Sample                   := 16,
           Dat_err                  := #err_uzloulov_in,
           Dat_f                    := "COM".dPr_uzloulov_in,
           Dat_md                   := MD 4200);
      NOP   0;
NETWORK
TITLE = НЯ Датчик тиску Млин ДМ-2 вхід
      CALL  "Dat_Filt" , DB 152 (
           dPIW                     := "dMlyn_in",
           dHi_lim                  := MD 3408,
           dLow_lim                 := MD 3412,
           dErr_lvl                 := -300,
           Sample                   := 16,
           Dat_err                  := #err_dMlyn_in,
           Dat_f                    := "COM".dMlyn_in,
           Dat_md                   := MD 4204);
      NOP   0;
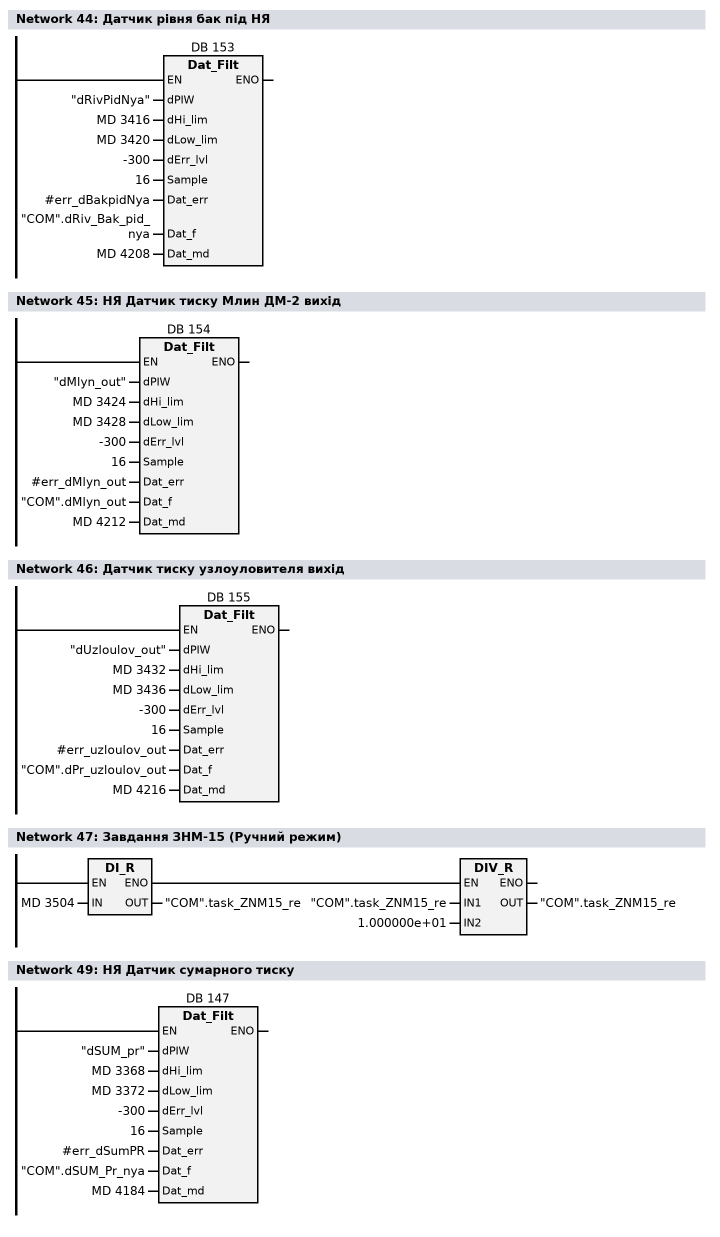
NETWORK
TITLE = Датчик рівня бак під НЯ
      CALL  "Dat_Filt" , DB 153 (
           dPIW                     := "dRivPidNya",
           dHi_lim                  := MD 3416,
           dLow_lim                 := MD 3420,
           dErr_lvl                 := -300,
           Sample                   := 16,
           Dat_err                  := #err_dBakpidNya,
           Dat_f                    := "COM".dRiv_Bak_pid_nya,
           Dat_md                   := MD 4208);
      NOP   0;
NETWORK
TITLE = НЯ Датчик тиску Млин ДМ-2 вихід
      CALL  "Dat_Filt" , DB 154 (
           dPIW                     := "dMlyn_out",
           dHi_lim                  := MD 3424,
           dLow_lim                 := MD 3428,
           dErr_lvl                 := -300,
           Sample                   := 16,
           Dat_err                  := #err_dMlyn_out,
           Dat_f                    := "COM".dMlyn_out,
           Dat_md                   := MD 4212);
      NOP   0;
NETWORK
TITLE = Датчик тиску узлоуловителя вихід
      CALL  "Dat_Filt" , DB 155 (
           dPIW                     := "dUzloulov_out",
           dHi_lim                  := MD 3432,
           dLow_lim                 := MD 3436,
           dErr_lvl                 := -300,
           Sample                   := 16,
           Dat_err                  := #err_uzloulov_out,
           Dat_f                    := "COM".dPr_uzloulov_out,
           Dat_md                   := MD 4216);
      NOP   0;
NETWORK
TITLE = Завдання ЗНМ-15 (Ручний режим)
//*****************  Завдання ЗНМ-15 в real ***********************************
      A(;
      L     MD 3504;
      DTR;
      T     "COM".task_ZNM15_re;
      SET;
      SAVE;
      CLR;
      A     BR;
      );
      JNB   _003;
      L     "COM".task_ZNM15_re;
      L     1.000000e+01;
      /R;
      T     "COM".task_ZNM15_re;
_003: NOP   0;
NETWORK
TITLE = Завдання ЗНМ-15 записуємо в AO 1_3 (ручний режим)
      A(;
      A     #bipolar;
      =     L 33.0;
      BLD   103;
      A     "ZNM15_HM";
      JNB   _004;
      CALL  "UNSCALE" (
           $1                       := "COM".task_ZNM15_re,
           $2                       := L#1120403456,
           $3                       := L#0,
           $4                       := L 33.0,
           $5                       := #ZNM15_ret,
           $6                       := P#M 4504.0);
_004: A     BR;
      );
      JNB   _005;
      L     MW 4504;
      T     "taskZNM15";
_005: NOP   0;
NETWORK
TITLE = НЯ Датчик сумарного тиску
//НЯ Датчик сумарного тиску
      CALL  "Dat_Filt" , DB 147 (
           dPIW                     := "dSUM_pr",
           dHi_lim                  := MD 3368,
           dLow_lim                 := MD 3372,
           dErr_lvl                 := -300,
           Sample                   := 16,
           Dat_err                  := #err_dSumPR,
           Dat_f                    := "COM".dSUM_Pr_nya,
           Dat_md                   := MD 4184);
      NOP   0;
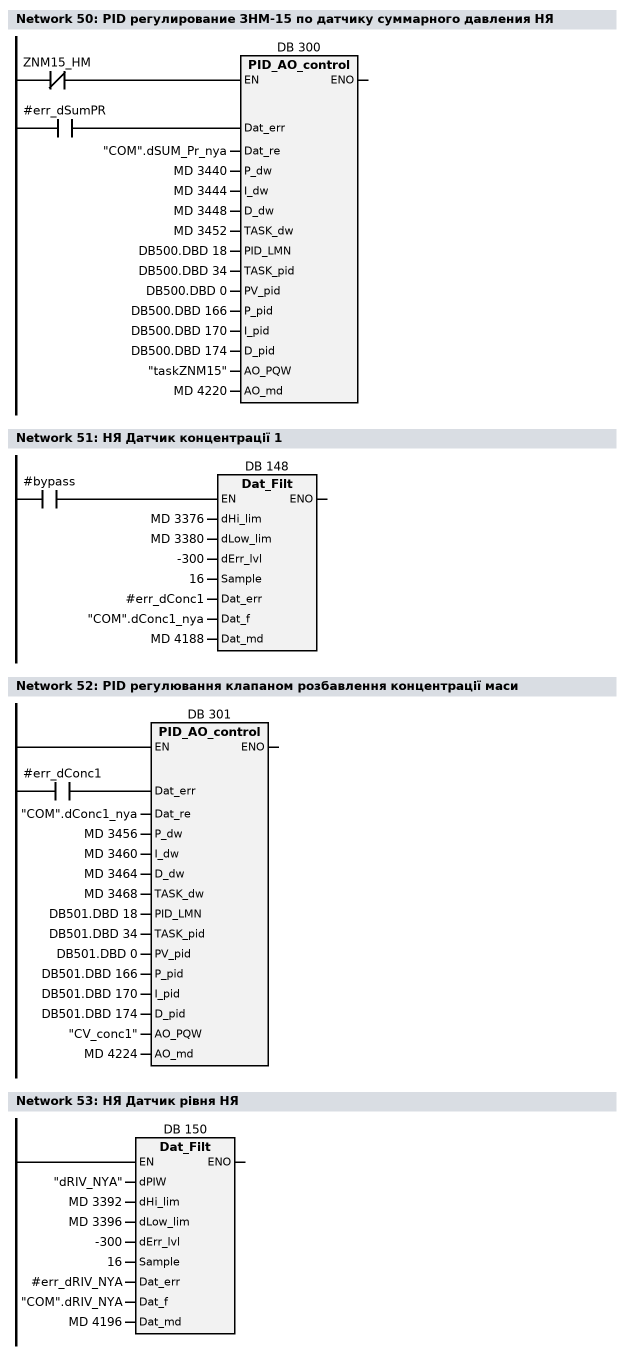
NETWORK
TITLE = PID регулирование ЗНМ-15 по датчику суммарного давления НЯ
//PID регулирование ЗНМ-15 по датчику суммарного давления НЯ
      A     #err_dSumPR;
      =     L 33.0;
      BLD   103;
      AN    "ZNM15_HM";
      JNB   _006;
      CALL  "PID_AO_control" , DB 300 (
           Dat_err                  := L 33.0,
           Dat_re                   := "COM".dSUM_Pr_nya,
           P_dw                     := MD 3440,
           I_dw                     := MD 3444,
           D_dw                     := MD 3448,
           TASK_dw                  := MD 3452,
           PID_LMN                  := DB500.DBD 18,
           TASK_pid                 := DB500.DBD 34,
           PV_pid                   := DB500.DBD 0,
           P_pid                    := DB500.DBD 166,
           I_pid                    := DB500.DBD 170,
           D_pid                    := DB500.DBD 174,
           AO_PQW                   := "taskZNM15",
           AO_md                    := MD 4220);
_006: NOP   0;
NETWORK
TITLE = НЯ Датчик концентрації 1
//НЯ Датчик концентрації1 (не підключений)
      A     #bypass;
      JNB   _007;
      CALL  "Dat_Filt" , DB 148 (
           dHi_lim                  := MD 3376,
           dLow_lim                 := MD 3380,
           dErr_lvl                 := -300,
           Sample                   := 16,
           Dat_err                  := #err_dConc1,
           Dat_f                    := "COM".dConc1_nya,
           Dat_md                   := MD 4188);
_007: NOP   0;
NETWORK
TITLE = PID регулювання клапаном розбавлення концентрації маси
      A     #err_dConc1;
      =     L 33.0;
      BLD   103;
      CALL  "PID_AO_control" , DB 301 (
           Dat_err                  := L 33.0,
           Dat_re                   := "COM".dConc1_nya,
           P_dw                     := MD 3456,
           I_dw                     := MD 3460,
           D_dw                     := MD 3464,
           TASK_dw                  := MD 3468,
           PID_LMN                  := DB501.DBD 18,
           TASK_pid                 := DB501.DBD 34,
           PV_pid                   := DB501.DBD 0,
           P_pid                    := DB501.DBD 166,
           I_pid                    := DB501.DBD 170,
           D_pid                    := DB501.DBD 174,
           AO_PQW                   := "CV_conc1",
           AO_md                    := MD 4224);
      NOP   0;
NETWORK
TITLE = НЯ Датчик рівня НЯ
      CALL  "Dat_Filt" , DB 150 (
           dPIW                     := "dRIV_NYA",
           dHi_lim                  := MD 3392,
           dLow_lim                 := MD 3396,
           dErr_lvl                 := -300,
           Sample                   := 16,
           Dat_err                  := #err_dRIV_NYA,
           Dat_f                    := "COM".dRIV_NYA,
           Dat_md                   := MD 4196);
      NOP   0;
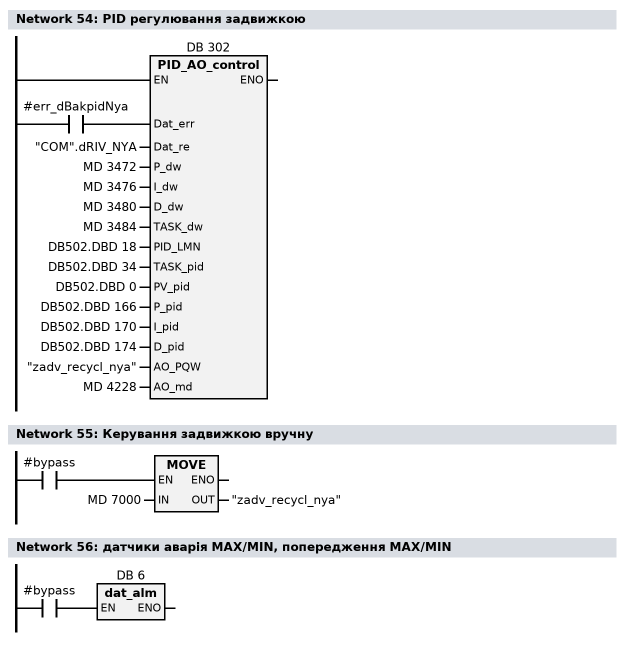
NETWORK
TITLE = PID регулювання задвижкою
      A     #err_dBakpidNya;
      =     L 33.0;
      BLD   103;
      CALL  "PID_AO_control" , DB 302 (
           Dat_err                  := L 33.0,
           Dat_re                   := "COM".dRIV_NYA,
           P_dw                     := MD 3472,
           I_dw                     := MD 3476,
           D_dw                     := MD 3480,
           TASK_dw                  := MD 3484,
           PID_LMN                  := DB502.DBD 18,
           TASK_pid                 := DB502.DBD 34,
           PV_pid                   := DB502.DBD 0,
           P_pid                    := DB502.DBD 166,
           I_pid                    := DB502.DBD 170,
           D_pid                    := DB502.DBD 174,
           AO_PQW                   := "zadv_recycl_nya",
           AO_md                    := MD 4228);
      NOP   0;
NETWORK
TITLE = Керування задвижкою вручну
      A     #bypass;
      JNB   _008;
      L     MD 7000;
      T     "zadv_recycl_nya";
_008: NOP   0;
NETWORK
TITLE = датчики аварія MAX/MIN, попередження MAX/MIN
      A     #bypass;
      JNB   _009;
      CALL  "dat_alm" , DB 6;
_009: NOP   0;
END_ORGANIZATION_BLOCK

ORGANIZATION_BLOCK "CYC_INT5"	// OB 35
TITLE = "Cyclic Interrupt"
VERSION : 0.1
VAR_TEMP
  OB35_EV_CLASS : BYTE ;	//Bits 0-3 = 1 (Coming event), Bits 4-7 = 1 (Event class 1)
  OB35_STRT_INF : BYTE ;	//16#36 (OB 35 has started)
  OB35_PRIORITY : BYTE ;	//Priority of OB Execution
  OB35_OB_NUMBR : BYTE ;	//35 (Organization block 35, OB35)
  OB35_RESERVED_1 : BYTE ;	//Reserved for system
  OB35_RESERVED_2 : BYTE ;	//Reserved for system
  OB35_PHASE_OFFSET : WORD ;	//Phase offset (msec)
  OB35_RESERVED_3 : INT ;	//Reserved for system
  OB35_EXC_FREQ : INT ;	//Frequency of execution (msec)
  OB35_DATE_TIME : DATE_AND_TIME ;	//Date and time OB35 started
  manual : BOOL ;
END_VAR
BEGIN
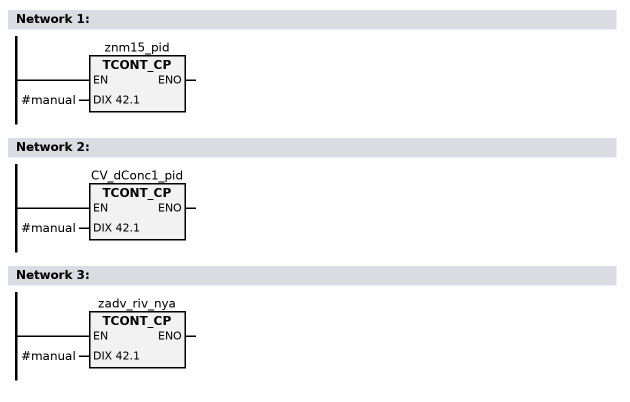
NETWORK
TITLE =
      CALL  "TCONT_CP" , "znm15_pid" (
           DIX 42.1                 := #manual);
      NOP   0;
NETWORK
TITLE =
      CALL  "TCONT_CP" , "CV_dConc1_pid" (
           DIX 42.1                 := #manual);
      NOP   0;
NETWORK
TITLE =
      CALL  "TCONT_CP" , "zadv_riv_nya" (
           DIX 42.1                 := #manual);
      NOP   0;
END_ORGANIZATION_BLOCK
